TYPE stData :
STRUCT
	iId: LINT;
	bSync: BOOL;
	dtTimestamp: DT;
	rSpeed: LREAL;
	rPos: LREAL;
	bPulse: BOOL;
END_STRUCT
END_TYPE

(* stored: Version 1.1.0.1, ProductVersion 3.1.4024.4
   DUT stData: Id {03f0b184-78c7-4813-83bd-dff7bb2e75b2} *)
